FUNCTION NewMessage : ST_Message
VAR_INPUT
	eMessage : E_MessageList;
	ePeer : E_PeersList;
END_VAR
VAR
END_VAR

NewMessage.eMessage := eMessage;
NewMessage.ePeer := ePeer;

END_FUNCTION

(* stored: Version 1.1.0.1, ProductVersion 3.1.4022.12
   POU NewMessage: Id {ec0e6791-e369-4a98-a9a5-8239f1aa4efc}, SpecialFunc None *)
